TYPE sMqttOut :
STRUCT
	sError: sError;
	sJobState: sJobState;
	sGeneralState: sGeneralState;
	sToken: sToken;
END_STRUCT
END_TYPE

(* stored: Version 1.1.0.1, ProductVersion 3.1.4026.13
   DUT sMqttOut: Id {9303d083-53b0-4c66-a65a-b0d4ee4a5e1f} *)
